(* CODESYS project EX4.project

Project tree, tasks and I/O mapping:
  Device : CODESYS Control Win V3, 3S - Smart Software Solutions GmbH, order no. 305021, version 3.5.11.30
    application Application
      libraries: Standard, * (System)
      task MainTask (cyclic, interval t#20ms, priority 1) calls PLC_PRG
      program PLC_PRG [LD]
*)

// Device/Application/PLC_PRG
PROGRAM PLC_PRG
VAR
	KM2: BOOL;       // CONTATOR DO MOTOR 2
	KM3: BOOL;       // CONTATOR DO MOTOR 3
	KM0: BOOL;       // SENTIDO REVERSO DO MOTOR 1
	KM1 : BOOL;      // SENTIDO DIRETO DE MOTOR 1
	SENSOR : BOOL;   // SENSOR DA MESA DO OPERADOR
	STOP : BOOL;     // PARA TUDO
	P1: BOOL;        // PASSO 1
	P2: BOOL;        // PASSO 2
	P3: BOOL;        // PASSO 3
	P4 : BOOL;       // INDICA QUE CHEGOU EM M3 E COMEÇA O PAÇO 4
	P5: BOOL;        // PASSO5
	P6: BOOL;        // PASSO 6
	TOF_1: TOF;
	ET1: TIME;
	TOF_2: TOF;
	ET2: TIME;;
	RETIRA_PECA: BOOL;
	AUX_KM1: BOOL;
	MESA_OPERA: BOOL;
	SISTEMA: BOOL;
	PARA: BOOL;
	FC3: BOOL;
	FC2: BOOL;
END_VAR
VAR // added by the converter: edge detectors and wires of the graphical bodies
    _rt1, _rt2 : R_TRIG;
END_VAR

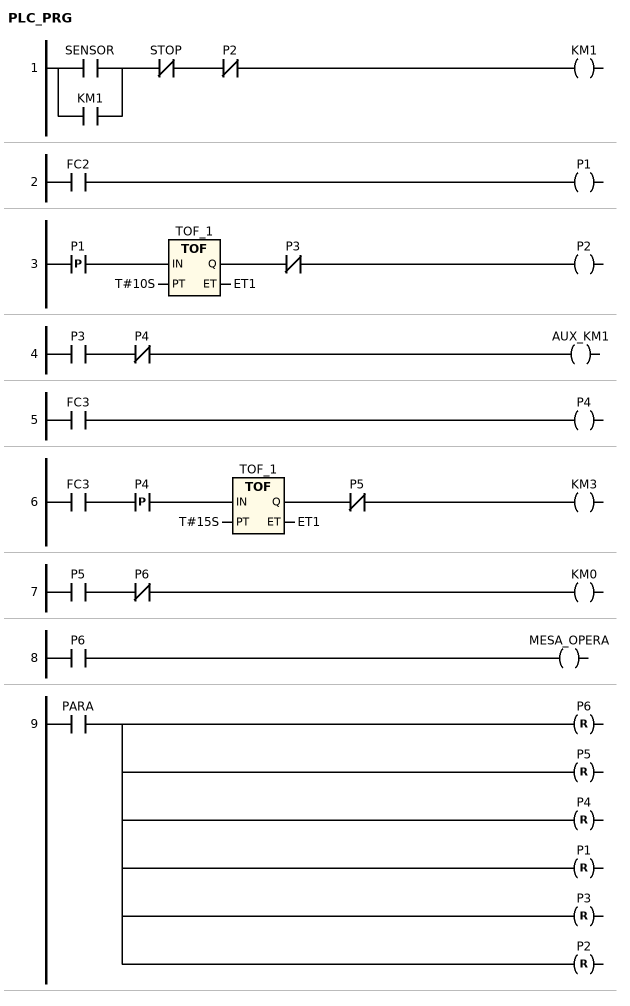
// NETWORK 1
KM1 := (SENSOR OR KM1) AND NOT STOP AND NOT P2;

// NETWORK 2
P1 := FC2;

// NETWORK 3
_rt1(CLK := P1);
TOF_1(IN := _rt1.Q, PT := T#10S, ET => ET1); // TOF
P2 := TOF_1.Q AND NOT P3;

// NETWORK 4
AUX_KM1 := P3 AND NOT P4;

// NETWORK 5
P4 := FC3;

// NETWORK 6
_rt2(CLK := P4);
TOF_1(IN := FC3 AND _rt2.Q, PT := T#15S, ET => ET1); // TOF
KM3 := TOF_1.Q AND NOT P5;

// NETWORK 7
KM0 := P5 AND NOT P6;

// NETWORK 8
MESA_OPERA := P6;

// NETWORK 9
P6 R= PARA;
P5 R= PARA;
P4 R= PARA;
P1 R= PARA;
P3 R= PARA;
P2 R= PARA;

END_PROGRAM
